FUNCTION_BLOCK AUDI_UDINT_AX_SEL_AUDI (* binary selection *)
  (* Standard: 61499-2; Description: Copyright (c) 2026 HR Agrartechnik GmbH This program and the accompanying materials are made available under the terms of the Eclipse Public License 2.0 which is available at https://www.eclipse.org/legal/epl-2.0/ SPDX-License-Identifier: EPL-2.0 *)
  (* Version 1.0, 2026-04-19, Franz Höpfinger, HR Agrartechnik GmbH, initial API and implementation *)
  PACKAGE adapter::iec61131::selection;
  IMPORT eclipse4diac::core::TypeHash;
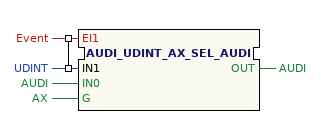
  EVENT_INPUT
    EI1 WITH IN1; (* Set IN1 *)
  END_EVENT
  VAR_INPUT
    IN1 : UDINT; (* Selectable input variable *)
  END_VAR
  SOCKETS
    IN0 : adapter::types::unidirectional::AUDI; (* Selectable input variable *)
    G : adapter::types::unidirectional::AX; (* Selector *)
  END_SOCKETS
  PLUGS
    OUT : adapter::types::unidirectional::AUDI; (* Selected Output *)
  END_PLUGS
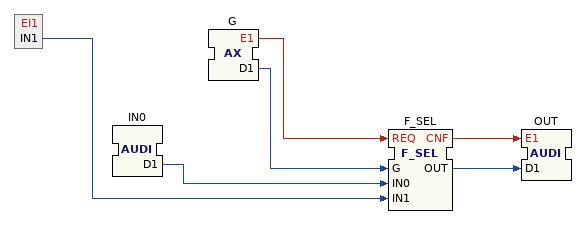
  FBS
    F_SEL : iec61131::selection::F_SEL;
  END_FBS
  EVENT_CONNECTIONS
    F_SEL.CNF TO OUT.E1;
    G.E1 TO F_SEL.REQ;
  END_CONNECTIONS
  DATA_CONNECTIONS
    F_SEL.OUT TO OUT.D1;
    G.D1 TO F_SEL.G;
    IN0.D1 TO F_SEL.IN0;
    IN1 TO F_SEL.IN1;
  END_CONNECTIONS
END_FUNCTION_BLOCK
